FUNCTION_BLOCK Aborted IMPLEMENTS ITF_PackMLState
VAR
END_VAR

METHOD CyclicLogic : BOOL
VAR_INPUT
END_VAR
END_METHOD

{warning 'add method implementation '}
METHOD EStop : BOOL
END_METHOD

{warning 'add method implementation '}
METHOD Reset : BOOL
END_METHOD

{warning 'add method implementation '}
METHOD Start : BOOL
END_METHOD

{warning 'add method implementation '}
METHOD Stop : BOOL
END_METHOD

END_FUNCTION_BLOCK

(* stored: Version 1.1.0.1, ProductVersion 3.1.4024.12
   POU Aborted: Id {9d11f351-b4bf-4f98-a02b-044980c0fcf0}, SpecialFunc None
   Method CyclicLogic: Id {f22e22e5-54e6-4715-a83e-723d936743bd}
   Method EStop: Id {1c038dc6-38e7-4546-b25e-01963f2585e2}
   Method Reset: Id {cb08e04f-e3a3-4729-87b7-21953aad123b}
   Method Start: Id {94432c27-b53a-49a2-90e2-527d66d45328}
   Method Stop: Id {4be6a551-e4c1-49cc-83c1-f9278ebab854} *)
